LIN {X 0,Y 53.352,Z 554.369,A -85,B 0,C 180,E1 -30397.237,E2 -30397.237} C_VEL
LIN {X 0,Y 62.213,Z 548.788,A -85,B 0,C 180,E1 -30403.788,E2 -30403.788} C_VEL
LIN {X 0,Y 71.488,Z 541.732,A -85,B 0,C 180,E1 -30409.455,E2 -30409.455} C_VEL
LIN {X 0,Y 73.263,Z 540.069,A -85,B 0,C 180,E1 -30410.914,E2 -30410.914} C_VEL
LIN {X 0,Y 74.589,Z 538.062,A -85,B 0,C 180,E1 -30414.594,E2 -30414.594} C_VEL
LIN {X 0,Y 75.296,Z 536.823,A -85,B 0,C 180,E1 -30417.325,E2 -30417.325} C_VEL
LIN {X 0,Y 75.751,Z 535.906,A -85,B 0,C 180,E1 -30420,E2 -30420} C_VEL
LIN {X 0,Y 74.885,Z 535.821,A -85,B 0,C 180,E1 -30425.385,E2 -30425.385} C_VEL
LIN {X 0,Y 73.699,Z 536.396,A -85,B 0,C 180,E1 -30430.995,E2 -30430.995} C_VEL
LIN {X 0,Y 72.049,Z 537.773,A -85,B 0,C 180,E1 -30437.016,E2 -30437.016} C_VEL
LIN {X 0,Y 71.323,Z 538.503,A -85,B 0,C 180,E1 -30440.135,E2 -30440.135} C_VEL
LIN {X 0,Y 69.181,Z 540.279,A -85,B 0,C 180,E1 -30443.892,E2 -30443.892} C_VEL
LIN {X 0,Y 60.273,Z 545.632,A -85,B 0,C 180,E1 -30449.01,E2 -30449.01} C_VEL
LIN {X 0,Y 51.73,Z 549.866,A -85,B 0,C 180,E1 -30455.395,E2 -30455.395} C_VEL
LIN {X 0,Y 46.479,Z 552.097,A -85,B 0,C 180,E1 -30460.882,E2 -30460.882} C_VEL
LIN {X 0,Y 41.673,Z 553.914,A -85,B 0,C 180,E1 -30467.576,E2 -30467.576} C_VEL
LIN {X 0,Y 37.516,Z 555.277,A -85,B 0,C 180,E1 -30475.805,E2 -30475.805} C_VEL
LIN {X 0,Y 32.459,Z 556.792,A -85,B 0,C 180,E1 -30497.494,E2 -30497.494} C_VEL
LIN {X 0,Y 31.77,Z 557.007,A -85,B 0,C 180,E1 -30509.999,E2 -30509.999} C_VEL
LIN {X 0,Y 32.457,Z 556.815,A -85,B 0,C 180,E1 -30522.504,E2 -30522.504} C_VEL
LIN {X 0,Y 37.504,Z 555.332,A -85,B 0,C 180,E1 -30544.206,E2 -30544.206} C_VEL
LIN {X 0,Y 41.655,Z 553.994,A -85,B 0,C 180,E1 -30552.443,E2 -30552.443} C_VEL
LIN {X 0,Y 49.078,Z 551.161,A -85,B 0,C 180,E1 -30561.961,E2 -30561.961} C_VEL
LIN {X 0,Y 57.363,Z 547.333,A -85,B 0,C 180,E1 -30569.05,E2 -30569.05} C_VEL
LIN {X 0,Y 67.745,Z 541.39,A -85,B 0,C 180,E1 -30575.482,E2 -30575.482} C_VEL
LIN {X 0,Y 69.16,Z 540.484,A -85,B 0,C 180,E1 -30576.144,E2 -30576.144} C_VEL
LIN {X 0,Y 71.369,Z 538.686,A -85,B 0,C 180,E1 -30579.899,E2 -30579.899} C_VEL
LIN {X 0,Y 72.728,Z 537.413,A -85,B 0,C 180,E1 -30585.09,E2 -30585.09} C_VEL
LIN {X 0,Y 73.714,Z 536.62,A -85,B 0,C 180,E1 -30589.007,E2 -30589.007} C_VEL
LIN {X 0,Y 74.923,Z 536.044,A -85,B 0,C 180,E1 -30594.617,E2 -30594.617} C_VEL
LIN {X 0,Y 75.769,Z 536.143,A -85,B 0,C 180,E1 -30600,E2 -30600} C_VEL
LIN {X 0,Y 74.739,Z 538.187,A -85,B 0,C 180,E1 -30605.395,E2 -30605.395} C_VEL
LIN {X 0,Y 73.365,Z 540.236,A -85,B 0,C 180,E1 -30609.131,E2 -30609.131} C_VEL
LIN {X 0,Y 71.505,Z 541.966,A -85,B 0,C 180,E1 -30610.622,E2 -30610.622} C_VEL
LIN {X 0,Y 66.721,Z 545.703,A -85,B 0,C 180,E1 -30613.39,E2 -30613.39} C_VEL
LIN {X 0,Y 62.2,Z 548.745,A -85,B 0,C 180,E1 -30615.51,E2 -30615.51} C_VEL
LIN {X 0,Y 57.123,Z 551.47,A -85,B 0,C 180,E1 -30616.991,E2 -30616.991} C_VEL
LIN {X 0,Y 46.252,Z 556.035,A -85,B 0,C 180,E1 -30619.815,E2 -30619.815} C_VEL
LIN {X 0,Y 40.956,Z 557.983,A -85,B 0,C 180,E1 -30622.574,E2 -30622.574} C_VEL
LIN {X 0,Y 39.311,Z 558.589,A -85,B 0,C 180,E1 -30623.953,E2 -30623.953} C_VEL
LIN {X 0,Y 32.995,Z 560.856,A -85,B 0,C 180,E1 -30631.57,E2 -30631.57} C_VEL
LIN {X 0,Y 24.392,Z 563.599,A -85,B 0,C 180,E1 -30654.814,E2 -30654.814} C_VEL
LIN {X 0,Y 22.449,Z 564.395,A -85,B 0,C 180,E1 -30671.757,E2 -30671.757} C_VEL
LIN {X 0,Y 22.603,Z 564.783,A -85,B 0,C 180,E1 -30690.001,E2 -30690.001} C_VEL
LIN {X 0,Y 24.383,Z 563.564,A -85,B 0,C 180,E1 -30725.204,E2 -30725.204} C_VEL
LIN {X 0,Y 32.987,Z 560.786,A -85,B 0,C 180,E1 -30748.455,E2 -30748.455} C_VEL
LIN {X 0,Y 41.644,Z 557.602,A -85,B 0,C 180,E1 -30758.159,E2 -30758.159} C_VEL
LIN {X 0,Y 50.96,Z 553.316,A -85,B 0,C 180,E1 -30764.886,E2 -30764.886} C_VEL
LIN {X 0,Y 60.54,Z 547.707,A -85,B 0,C 180,E1 -30770.666,E2 -30770.666} C_VEL
LIN {X 0,Y 66.968,Z 543.259,A -85,B 0,C 180,E1 -30773.976,E2 -30773.976} C_VEL
LIN {X 0,Y 69.04,Z 541.263,A -85,B 0,C 180,E1 -30777.083,E2 -30777.083} C_VEL
LIN {X 0,Y 69.791,Z 540.2,A -85,B 0,C 180,E1 -30780,E2 -30780} C_VEL
LIN {X 0,Y 68.841,Z 540.05,A -85,B 0,C 180,E1 -30785.86,E2 -30785.86} C_VEL
LIN {X 0,Y 67.283,Z 540.747,A -85,B 0,C 180,E1 -30792.059,E2 -30792.059} C_VEL
LIN {X 0,Y 65.973,Z 541.607,A -85,B 0,C 180,E1 -30796.51,E2 -30796.51} C_VEL
LIN {X 0,Y 64.833,Z 542.386,A -85,B 0,C 180,E1 -30798.978,E2 -30798.978} C_VEL
LIN {X 0,Y 60.309,Z 544.993,A -85,B 0,C 180,E1 -30801.208,E2 -30801.208} C_VEL
LIN {X 0,Y 51.031,Z 549.582,A -85,B 0,C 180,E1 -30806.466,E2 -30806.466} C_VEL
LIN {X 0,Y 42.215,Z 553.103,A -85,B 0,C 180,E1 -30813.652,E2 -30813.652} C_VEL
LIN {X 0,Y 36.792,Z 554.92,A -85,B 0,C 180,E1 -30820.172,E2 -30820.172} C_VEL
LIN {X 0,Y 31.948,Z 556.283,A -85,B 0,C 180,E1 -30828.703,E2 -30828.703} C_VEL
LIN {X 0,Y 25.643,Z 557.797,A -85,B 0,C 180,E1 -30854.092,E2 -30854.092} C_VEL
LIN {X 0,Y 24.742,Z 558.012,A -85,B 0,C 180,E1 -30869.999,E2 -30869.999} C_VEL
LIN {X 0,Y 25.641,Z 557.82,A -85,B 0,C 180,E1 -30885.907,E2 -30885.907} C_VEL
LIN {X 0,Y 31.937,Z 556.336,A -85,B 0,C 180,E1 -30911.312,E2 -30911.312} C_VEL
LIN {X 0,Y 36.776,Z 554.998,A -85,B 0,C 180,E1 -30919.853,E2 -30919.853} C_VEL
LIN {X 0,Y 45.088,Z 552.166,A -85,B 0,C 180,E1 -30929.013,E2 -30929.013} C_VEL
LIN {X 0,Y 54.086,Z 548.337,A -85,B 0,C 180,E1 -30935.448,E2 -30935.448} C_VEL
LIN {X 0,Y 64.821,Z 542.589,A -85,B 0,C 180,E1 -30941.018,E2 -30941.018} C_VEL
LIN {X 0,Y 65.993,Z 541.79,A -85,B 0,C 180,E1 -30943.427,E2 -30943.427} C_VEL
LIN {X 0,Y 67.324,Z 540.932,A -85,B 0,C 180,E1 -30947.949,E2 -30947.949} C_VEL
LIN {X 0,Y 68.857,Z 540.248,A -85,B 0,C 180,E1 -30954.141,E2 -30954.141} C_VEL
LIN {X 0,Y 69.795,Z 540.417,A -85,B 0,C 180,E1 -30960,E2 -30960} C_VEL
LIN {X 0,Y 69.123,Z 541.413,A -85,B 0,C 180,E1 -30962.914,E2 -30962.914} C_VEL
LIN {X 0,Y 67.091,Z 543.382,A -85,B 0,C 180,E1 -30966.013,E2 -30966.013} C_VEL
LIN {X 0,Y 57.314,Z 549.875,A -85,B 0,C 180,E1 -30971.196,E2 -30971.196} C_VEL
LIN {X 0,Y 48.35,Z 554.744,A -85,B 0,C 180,E1 -30976.9,E2 -30976.9} C_VEL
LIN {X 0,Y 39.311,Z 558.589,A -85,B 0,C 180,E1 -30983.953,E2 -30983.953} C_VEL
LIN {X 0,Y 34.343,Z 560.201,A -85,B 0,C 180,E1 -30988.265,E2 -30988.265} C_VEL
LIN {X 0,Y 25.554,Z 562.031,A -85,B 0,C 180,E1 -30996.379,E2 -30996.379} C_VEL
LIN {X 0,Y 19.084,Z 562.931,A -85,B 0,C 180,E1 -31008.138,E2 -31008.138} C_VEL
LIN {X 0,Y 15.831,Z 563.401,A -85,B 0,C 180,E1 -31024.423,E2 -31024.423} C_VEL
LIN {X 0,Y 15.353,Z 563.49,A -85,B 0,C 180,E1 -31031.449,E2 -31031.449} C_VEL
LIN {X 0,Y 15.447,Z 563.76,A -85,B 0,C 180,E1 -31050.002,E2 -31050.002} C_VEL
LIN {X 0,Y 15.952,Z 563.3,A -85,B 0,C 180,E1 -31078.224,E2 -31078.224} C_VEL
LIN {X 0,Y 23.971,Z 561.349,A -85,B 0,C 180,E1 -31111.594,E2 -31111.594} C_VEL
LIN {X 0,Y 33.022,Z 558.786,A -85,B 0,C 180,E1 -31123.287,E2 -31123.287} C_VEL
LIN {X 0,Y 42.866,Z 555.257,A -85,B 0,C 180,E1 -31129.655,E2 -31129.655} C_VEL
LIN {X 0,Y 49.549,Z 552.257,A -85,B 0,C 180,E1 -31133.169,E2 -31133.169} C_VEL
LIN {X 0,Y 59.782,Z 546.624,A -85,B 0,C 180,E1 -31137.834,E2 -31137.834} C_VEL
LIN {X 0,Y 62.271,Z 545.039,A -85,B 0,C 180,E1 -31138.86,E2 -31138.86} C_VEL
LIN {X 0,Y 63.372,Z 544.224,A -85,B 0,C 180,E1 -31140,E2 -31140} C_VEL
LIN {X 0,Y 63.299,Z 543.946,A -85,B 0,C 180,E1 -31142.192,E2 -31142.192} C_VEL
LIN {X 0,Y 62.418,Z 543.992,A -85,B 0,C 180,E1 -31146.465,E2 -31146.465} C_VEL
LIN {X 0,Y 60.421,Z 544.798,A -85,B 0,C 180,E1 -31153.453,E2 -31153.453} C_VEL
LIN {X 0,Y 58.137,Z 545.999,A -85,B 0,C 180,E1 -31154.737,E2 -31154.737} C_VEL
LIN {X 0,Y 48.31,Z 550.588,A -85,B 0,C 180,E1 -31158.983,E2 -31158.983} C_VEL
LIN {X 0,Y 38.765,Z 554.108,A -85,B 0,C 180,E1 -31164.972,E2 -31164.972} C_VEL
LIN {X 0,Y 32.702,Z 555.926,A -85,B 0,C 180,E1 -31170.721,E2 -31170.721} C_VEL
LIN {X 0,Y 27.068,Z 557.288,A -85,B 0,C 180,E1 -31178.836,E2 -31178.836} C_VEL
LIN {X 0,Y 18.982,Z 558.802,A -85,B 0,C 180,E1 -31208.267,E2 -31208.267} C_VEL
LIN {X 0,Y 17.714,Z 559.017,A -85,B 0,C 180,E1 -31229.998,E2 -31229.998} C_VEL
LIN {X 0,Y 18.98,Z 558.825,A -85,B 0,C 180,E1 -31251.731,E2 -31251.731} C_VEL
LIN {X 0,Y 27.059,Z 557.341,A -85,B 0,C 180,E1 -31281.185,E2 -31281.185} C_VEL
LIN {X 0,Y 32.689,Z 556.003,A -85,B 0,C 180,E1 -31289.312,E2 -31289.312} C_VEL
LIN {X 0,Y 41.906,Z 553.17,A -85,B 0,C 180,E1 -31297.279,E2 -31297.279} C_VEL
LIN {X 0,Y 51.563,Z 549.341,A -85,B 0,C 180,E1 -31302.57,E2 -31302.57} C_VEL
LIN {X 0,Y 58.109,Z 546.189,A -85,B 0,C 180,E1 -31305.366,E2 -31305.366} C_VEL
LIN {X 0,Y 60.451,Z 544.955,A -85,B 0,C 180,E1 -31306.554,E2 -31306.554} C_VEL
LIN {X 0,Y 62.429,Z 544.173,A -85,B 0,C 180,E1 -31313.536,E2 -31313.536} C_VEL
LIN {X 0,Y 63.298,Z 544.134,A -85,B 0,C 180,E1 -31317.817,E2 -31317.817} C_VEL
LIN {X 0,Y 63.454,Z 544.362,A -85,B 0,C 180,E1 -31320,E2 -31320} C_VEL
LIN {X 0,Y 62.312,Z 545.197,A -85,B 0,C 180,E1 -31321.118,E2 -31321.118} C_VEL
LIN {X 0,Y 52.928,Z 550.654,A -85,B 0,C 180,E1 -31325.207,E2 -31325.207} C_VEL
LIN {X 0,Y 42.866,Z 555.371,A -85,B 0,C 180,E1 -31330.355,E2 -31330.355} C_VEL
LIN {X 0,Y 33.026,Z 558.866,A -85,B 0,C 180,E1 -31336.746,E2 -31336.746} C_VEL
LIN {X 0,Y 23.974,Z 561.397,A -85,B 0,C 180,E1 -31348.425,E2 -31348.425} C_VEL
LIN {X 0,Y 15.812,Z 563.372,A -85,B 0,C 180,E1 -31383.612,E2 -31383.612} C_VEL
LIN {X 0,Y 15.353,Z 563.49,A -85,B 0,C 180,E1 -31391.449,E2 -31391.449} C_VEL
LIN {X 0,Y 14.495,Z 563.584,A -85,B 0,C 180,E1 -31403.331,E2 -31403.331} C_VEL
LIN {X 0,Y 12.777,Z 563.33,A -85,B 0,C 180,E1 -31421.424,E2 -31421.424} C_VEL
LIN {X 0,Y 12.599,Z 562.139,A -85,B 0,C 180,E1 -31466.224,E2 -31466.224} C_VEL
LIN {X 0,Y 15.335,Z 561.471,A -85,B 0,C 180,E1 -31478.848,E2 -31478.848} C_VEL
LIN {X 0,Y 28.264,Z 558.735,A -85,B 0,C 180,E1 -31494.065,E2 -31494.065} C_VEL
LIN {X 0,Y 38.671,Z 555.545,A -85,B 0,C 180,E1 -31498.328,E2 -31498.328} C_VEL
LIN {X 0,Y 46.101,Z 552.587,A -85,B 0,C 180,E1 -31500.724,E2 -31500.724} C_VEL
LIN {X 0,Y 56.365,Z 547.549,A -85,B 0,C 180,E1 -31504.04,E2 -31504.04} C_VEL
LIN {X 0,Y 56.424,Z 547.438,A -85,B 0,C 180,E1 -31504.821,E2 -31504.821} C_VEL
LIN {X 0,Y 55.597,Z 547.663,A -85,B 0,C 180,E1 -31507.263,E2 -31507.263} C_VEL
LIN {X 0,Y 52.815,Z 548.89,A -85,B 0,C 180,E1 -31508.934,E2 -31508.934} C_VEL
LIN {X 0,Y 43.094,Z 552.884,A -85,B 0,C 180,E1 -31511.891,E2 -31511.891} C_VEL
LIN {X 0,Y 36.36,Z 555.114,A -85,B 0,C 180,E1 -31514.882,E2 -31514.882} C_VEL
LIN {X 0,Y 29.732,Z 556.931,A -85,B 0,C 180,E1 -31518.996,E2 -31518.996} C_VEL
LIN {X 0,Y 23.313,Z 558.294,A -85,B 0,C 180,E1 -31525.255,E2 -31525.255} C_VEL
LIN {X 0,Y 12.722,Z 559.808,A -85,B 0,C 180,E1 -31556.464,E2 -31556.464} C_VEL
LIN {X 0,Y 10.686,Z 560.022,A -85,B 0,C 180,E1 -31589.997,E2 -31589.997} C_VEL
LIN {X 0,Y 12.72,Z 559.83,A -85,B 0,C 180,E1 -31623.535,E2 -31623.535} C_VEL
LIN {X 0,Y 23.306,Z 558.346,A -85,B 0,C 180,E1 -31654.775,E2 -31654.775} C_VEL
LIN {X 0,Y 29.723,Z 557.007,A -85,B 0,C 180,E1 -31661.045,E2 -31661.045} C_VEL
LIN {X 0,Y 39.724,Z 554.174,A -85,B 0,C 180,E1 -31666.671,E2 -31666.671} C_VEL
LIN {X 0,Y 49.911,Z 550.345,A -85,B 0,C 180,E1 -31670.291,E2 -31670.291} C_VEL
LIN {X 0,Y 52.805,Z 549.053,A -85,B 0,C 180,E1 -31671.157,E2 -31671.157} C_VEL
LIN {X 0,Y 55.606,Z 547.827,A -85,B 0,C 180,E1 -31672.739,E2 -31672.739} C_VEL
LIN {X 0,Y 56.423,Z 547.609,A -85,B 0,C 180,E1 -31675.187,E2 -31675.187} C_VEL
LIN {X 0,Y 56.363,Z 547.719,A -85,B 0,C 180,E1 -31675.968,E2 -31675.968} C_VEL
LIN {X 0,Y 46.092,Z 552.724,A -85,B 0,C 180,E1 -31679.282,E2 -31679.282} C_VEL
LIN {X 0,Y 38.671,Z 555.648,A -85,B 0,C 180,E1 -31681.711,E2 -31681.711} C_VEL
LIN {X 0,Y 28.265,Z 558.808,A -85,B 0,C 180,E1 -31685.974,E2 -31685.974} C_VEL
LIN {X 0,Y 15.126,Z 561.548,A -85,B 0,C 180,E1 -31701.681,E2 -31701.681} C_VEL
LIN {X 0,Y 8.42,Z 562.544,A -85,B 0,C 180,E1 -31745.113,E2 -31745.113} C_VEL
LIN {X 0,Y 8.299,Z 562.737,A -85,B 0,C 180,E1 -31770.004,E2 -31770.004} C_VEL
LIN {X 0,Y 9.906,Z 562.323,A -85,B 0,C 180,E1 -31815.194,E2 -31815.194} C_VEL
LIN {X 0,Y 15.335,Z 561.471,A -85,B 0,C 180,E1 -31838.848,E2 -31838.848} C_VEL
LIN {X 0,Y 15.2,Z 561.307,A -85,B 0,C 180,E1 -31842.729,E2 -31842.729} C_VEL
LIN {X 0,Y 13.566,Z 561.2,A -85,B 0,C 180,E1 -31848.24,E2 -31848.24} C_VEL
LIN {X 0,Y 9.952,Z 561.189,A -85,B 0,C 180,E1 -31857.465,E2 -31857.465} C_VEL
LIN {X 0,Y 3.605,Z 561.151,A -85,B 0,C 180,E1 -31901.442,E2 -31901.442} C_VEL
LIN {X 0,Y 4.599,Z 560.989,A -85,B 0,C 180,E1 -31989.893,E2 -31989.893} C_VEL
LIN {X 0,Y 6.057,Z 560.894,A -85,B 0,C 180,E1 -32003.524,E2 -32003.524} C_VEL
LIN {X 0,Y 14.426,Z 560.284,A -85,B 0,C 180,E1 -32026.987,E2 -32026.987} C_VEL
LIN {X 0,Y 14.145,Z 560.522,A -85,B 0,C 180,E1 -32033.566,E2 -32033.566} C_VEL
LIN {X 0,Y 6.162,Z 561.404,A -85,B 0,C 180,E1 -32039.997,E2 -32039.997} C_VEL
LIN {X 0,Y 1.155,Z 561.715,A -85,B 0,C 180,E1 -32130.029,E2 -32130.029} C_VEL
LIN {X 0,Y 12.897,Z 560.628,A -85,B 0,C 180,E1 -32225.986,E2 -32225.986} C_VEL
LIN {X 0,Y 14.146,Z 560.486,A -85,B 0,C 180,E1 -32226.46,E2 -32226.46} C_VEL
LIN {X 0,Y 14.428,Z 560.248,A -85,B 0,C 180,E1 -32233.031,E2 -32233.031} C_VEL
LIN {X 0,Y 7.886,Z 560.813,A -85,B 0,C 180,E1 -32246.97,E2 -32246.97} C_VEL
LIN {X 0,Y 6.057,Z 560.894,A -85,B 0,C 180,E1 -32363.524,E2 -32363.524} C_VEL
LIN {X 0,Y 7.794,Z 562.893,A -85,B 0,C 180,E1 -32372.686,E2 -32372.686} C_VEL
LIN {X 0,Y 7.794,Z 600,A -85,B 0,C 180,E1 -32372.686,E2 -32372.686} C_VEL
LIN {X 0,Y 7.794,Z 600,A -85,B 0,C 180,E1 -32372.686,E2 -32372.686}

QRS_NEXT_CUT()

QRS_NEXT()
QRS_HOME()

END
